// TIA Portal V18 export
DATA_BLOCK "Flowrate adjustment B"   // DB79
{ S7_Optimized_Access := 'TRUE' }
VERSION : 0.1
// stored: AutoNumber false, DBAccessibleFromOPCUA true, IsOnlyStoredInLoadMemory false, IsRetainMemResEnabled false, IsWriteProtectedInAS false, MemoryReserve 100
   VAR RETAIN
      percentage : Struct
         "5%" : Real;
         "10%" : Real;
         "15%" : Real;
         "20%" : Real;
         "25%" : Real;
         "30%" : Real;
         "40%" : Real;
         "50%" : Real;
         "60%" : Real;
         "70%" : Real;
         "80%" : Real;
         "90%" : Real;
         "100%" : Real;
      END_STRUCT;
   END_VAR
   VAR
      "Reset Flowadjustment B" : Bool;
   END_VAR
BEGIN
END_DATA_BLOCK
